RoboDK station: ROXS_2Robots.rdk

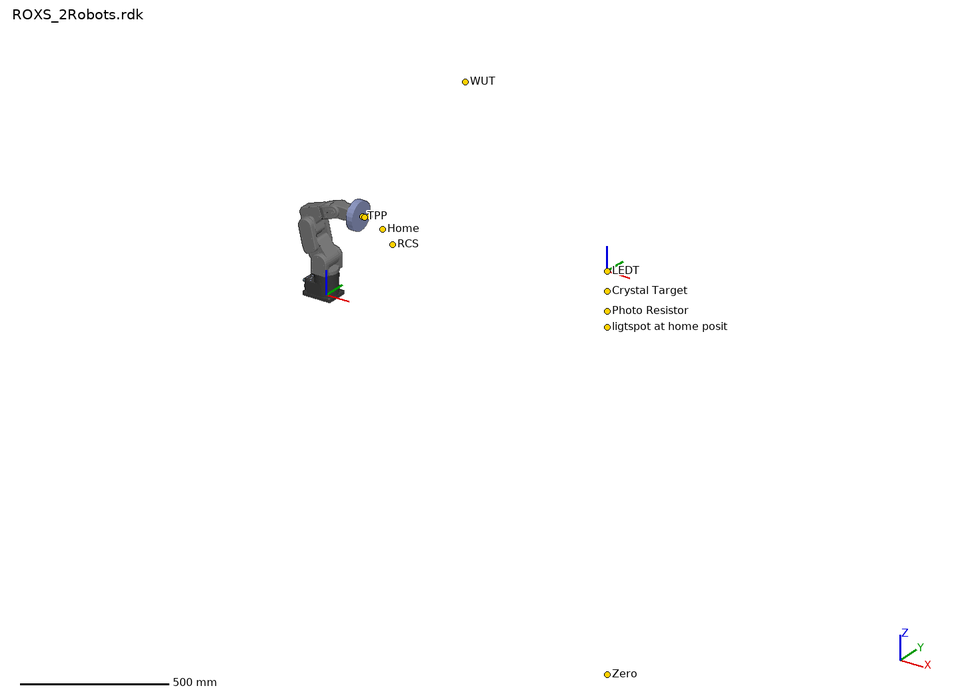
[picture v0: the station drawn from its stored meshes, robots at their saved joint values, targets as dots, program paths as lines]
Station ROXS_2Robots (saved by RoboDK 5.5.2). Poses are relative to the parent item; angles as X-Y-Z fixed-axis rotations.
  - frame LED at (0, 0, 0) mm
    - target Crystal Target (Cartesian target) at (0, 0, -75) mm; joints [-23.128, -26.053, 31.636, -77.168, -23.756, 166.237]
    - target ligtspot at home position (Cartesian target) at (0, 0, -209.55) mm; joints [0, 4.3, -4.481, 0, 0.181, 0]
    - target Zero (Cartesian target) at (0, 0, -1504.55) mm; joints [0, 0, 0, 0, 0, 0] of Mecademic Meca500 R3
    - target WUT (joint target) at (-822.96, 346.08, 338.94) mm, rotated rx -90 ry -86.86 rz -90 deg; joints [0, -22.866, 35.785, 0, -12.919, 0]
    - target Home (Cartesian target) at (-919.2, 0, -101.6) mm, rotated rx 0 ry 90 rz 0 deg; joints [0, 0, 0, 0, 0, 0] of Mecademic Meca500 R3
    - target Zoo wee mama (Cartesian target) at (-982, 12.9, -76.36) mm, rotated rx 0 ry 90 rz 0 deg; joints [12.714, -19.59, 2.794, -37.982, 20.954, -323.903] of Mecademic Meca500 R3
    - target RCS (Cartesian target) at (-950.17, 103.77, -207.82) mm, rotated rx 0 ry 90 rz -5.83 deg; joints [-142.099, -36.249, -124.258, 0, 70.507, -225.257] of Mecademic Meca500 R3
    - target LEDT (Cartesian target) at (0, 0, 0) mm, rotated rx 0 ry 90 rz -5.83 deg; joints [0, -33.951, 22.527, 0, 11.424, 0]
    - target Photo Resistor (Cartesian target) at (0, 0, -150) mm; joints [0, 0, 0, 0, 0, 0]
    - target TPP (Cartesian target) at (-1000, 0, -75) mm, rotated rx 0 ry 90 rz 0 deg; joints [71.078, 20.108, -37.888, -86.424, 78.994, -288.125] of Mecademic Meca500 R3
      - target Bing (Cartesian target) at (75, 0, 1000) mm; joints [0, -10.782, 3.761, 0, 7.021, -360] of Mecademic Meca500 R3
      - target APP (Cartesian target) at (1.62, 1.68, 7.33) mm; joints [0, -22.914, 36.46, 0, -13.546, 0] of Mecademic Meca500 R3
  - Python program Linear Move (listed below)
  - Python program Smart Spiral SSAP (listed below)
  - Python program Set Target Pos (listed below)
  - Python program R Scan (listed below)
  - frame Mecademic Meca500 R3 Base at (-1150, 1.09, -409.6) mm, rotated rx 0 ry 0 rz 0.06 deg
    - robot Mecademic Meca500 R3: 6 axes
        modified DH rows (alpha deg, a mm, theta deg, d mm): 0, 0, 0, 135; -90, 0, -90, 0; 0, 135, 0, 0; -90, 38, 0, 120; 90, 0, 0, 0; -90, 0, 180, 70
        joint limits [-175, -70, -135, -170, -115, -720] to [175, 90, 70, 170, 115, 720]; home [0, 0, 0, 0, 0, 0]; saved at [0.669, -23.965, 5.181, -2.263, 18.798, -357.858]
      - tool CrystalToolSample, TCP at (0, 0, 40.8) mm, size 107.9 x 25.4 x 107.9 mm, geometry from CrystalToolSample.STEP
  - Python program Prog15 (listed below)
  - Python program Prog16 (listed below)
  - Python program SetTarget2 (listed below)
  - Python program R Scan2 (listed below)

--- Python program Linear Move ---
from robodk.robolink import *       # import the robolink library (bridge with RoboDK)
from robodk.robomath import *       # import the robotics toolbox
RDK = Robolink()                    # establish a link with the simulator
robot = RDK.Item('Mecademic Meca500 R3')     # retrieve the robot by name




tool=RDK.Item('CrystalToolSample')
robot.setPoseTool(tool) # Update the TCP

robot.setSpeed(100)  # Set linear speed in mm/s
robot.setJoints([0,0,0,0,0,0])      # set all robot axes to zero



target = RDK.Item('TPP')         # retrieve the Target item
robot.MoveJ(target)                 # move the robot to the target


Final = target.Pose()*transl(0,20,0)
print(target.Pose())

rj=robot.Joints()

print(robot.MoveL_Test(rj,Final))

if robot.MoveL_Test(rj,Final) == 0:         # linear move to the approach position
    robot.MoveL(Final)


print('approach reached')
print('Attempting pose', Final)
#robot.MoveL(pose)

--- Python program Smart Spiral SSAP ---
"""
Created on Thu Jan 19 18:43:18 2023

@author: westj
"""
from robodk.robolink import *       # import the robolink library (bridge with RoboDK)
RDK = Robolink()
from robodk.robomath import *
import math
import numpy as np
import matplotlib.pyplot as plt
import array
import pandas as pd
import requests
import re
from scipy.signal import find_peaks, peak_prominences, savgol_filter
from scipy.stats import linregress
import json
import time
#******CLASSES AND CLASS FUNCTIONS****************************************************************************
class Spiral:
    def __init__(self,x0:float,y0:float,points:float) -> None:
        self.x0=x0 #x offset
        self.y0=y0 #y offset
        self.points=points

    def build(self, radius:float, spacing:float):
        revs=radius/spacing            #calc number of revolutions
        k=spacing/(2*np.pi)
        theta=np.array(np.linspace(0,revs*2*np.pi,self.points)) #how many points and angle coord
        r=k * theta                       #radius coord
        x=(r*np.cos(theta)+self.x0)       #convert to x cartesian
        y=(r*np.sin(theta)+self.y0)       #convert to y cartesian
        return x, y

class Linear:
    def __init__(self,data,points):
        self.data=data #data
        self.points=points #number of points to fit

    def get(self,x):
        peaks= find_peaks(self.data['Intensity'], prominence=[prominence],width=width,height=height)
        IPeaks=peaks[0]
        H=peaks[1]['peak_heights']
        A=[]
        for i in range(len(IPeaks)):
            corr=[IPeaks[i],H[i]]
            A.append(corr)
        SA=sorted(A, key=lambda x: x[1], reverse=True) #sort by peak height largest to smallest
        if len(SA) <= 1:

            E=np.sqrt((Ix-xl)**2+(Iy-yl)**2)
            print('***Linear Translation********************************************************')
            print(Ldata)
            print('_________SSAP Report:_________')
            print('Calculated peak is at',xl,yl)
            print('True peak is at',Ix,Iy)
            print('Error is:',E)
            print('Linear step size is:',step)
            raise Exception("Spiral did not find enough peaks")
        XPP=[]
        YPP=[]
        for i in range(self.points):
            #ICP.append(SA[i][0])
            XPP.append(self.data['X'][SA[i][0]])
            YPP.append(self.data['Y'][SA[i][0]])
        LRR=linregress(XPP,YPP)

        return LRR[0]*x+LRR[1]
    def getC(self,x,xl,yl):
        peaks= find_peaks(self.data['Intensity'], prominence=[prominence],width=width,height=height) #find peaks
        XPP=[xl]  #use origin of previous spiral as a point
        YPP=[yl]
        XPP.append(self.data['X'][peaks[0][0]])
        YPP.append(self.data['Y'][peaks[0][0]])
        LRR=linregress(XPP,YPP) #run regression
        return LRR[0]*x+LRR[1]


    def getSA(self):
        peaks= find_peaks(self.data['Intensity'],prominence=[prominence],width=width,height=height)
        IPeaks=peaks[0]
        H=peaks[1]['peak_heights']
        A=[]
        for i in range(len(IPeaks)):
            corr=[IPeaks[i],H[i]]
            A.append(corr)
        SA=sorted(A, key=lambda g: g[1], reverse=True) #sort by peak height largest to smallest
        return SA,IPeaks

class Webserver:
#webserver returns json string that looks like {"speed":25,"goalpos":140,"zCurrent":140.09935,"PRInt":4,"ledStatus":false,"zero":1}
    def __init__(self,IP,extenstion)->None:
        self.IP=IP #x offset
        self.ex=extenstion #y offset


    def patch(self, obj, value):
        url = "http://" + self.IP + "/" +self.ex #address of server
        obj=str(obj)

        payload = {obj: value} #rewrite the obj to value
        headers = {"Content-Type": "application/json"} #formatting the message as a json string don't change this

        response = requests.patch(url, data=json.dumps(payload), headers=headers) #patch in or change the value

        if response.status_code == 204: #if 204 which is http good patch
            print(obj + "Updated successfully")
        else:
            print(obj + "Error: ", response.status_code)
        return

    def get(self, obj):
        url = "http://" + self.IP + "/" +self.ex #address of server
        obj=str(obj)

        response = requests.get(url)
        if response.status_code == 200:
            value=response.json()[obj]
            print(obj, value)
        else:
           print("Error: ", response.status_code)

        return value


class Intensity: #intensity function is a gaussian curve
    def __init__(self,x0:float,y0:float, mu_x, mu_y, sigma_x, sigma_y):
        self.x0=-x0 #x offset
        self.y0=-y0 #y offset
        self.mu_x=mu_x
        self.mu_y=mu_y
        self.sigma_x=sigma_x #x squish/stretch
        self.sigma_y=sigma_y #y sqush/stretch


    def get(self,x, y): #gaussian curve definition
        I=np.exp(-0.5 * (((x +self.x0- self.mu_x) / self.sigma_x)**2 + ((y+self.y0 - self.mu_y) / self.sigma_y)**2))
        return I

class Photoresistor:
    def __init__(self,url) -> None:
        self.url=url
    def get(self):
        response = requests.get(self.url) #go to webserver under the url of the arduino/photoresistor
        if response.ok: #if we can connect
            value = response.text #screen scrape the web server
            pr=re.findall(r'\d+',value) #take the number off the webserver
            pri=-int(pr[0]) #reverse the sign of the number
            #print('Received value:', value)
            #print('Number', PR)
        else:
            print('Error:', response.status_code)


        return pri

#def Exit_SSAP(Intensity,plateau_size,height):
 #   if len(find_peaks(Intensity,plateau_size=pleatau_size,height=height)[0])>0:
    #    break

#***SPIRAL SCANNING ALIGNMENT PROCEDURE**************************************************************************************************************
#___Initialization______________
xl=0 #starting offset from target for spiral
yl=0
zl=0
Loops=3 #number of loops to run SSAP

robot = RDK.Item('Mecademic Meca500 R3') #define robot
home = RDK.Item('Home') #define robot home
target = RDK.Item('TPP')# retrieve the Target item

tool=RDK.Item('CrystalToolSample')
robot.setPoseTool(tool) # Update the TCP

PR= RDK.Item('Photo Resistor',ITEM_TYPE_TARGET)
X,Y,Z,A,B,C=Pose_2_KUKA(PR.Pose())

IP="192.168.0.99"
ext="values"
ESP=Webserver(IP,ext)

#robot.setSpeed(-1,75)
robot.setSpeed(100)  # Set linear speed in mm/s
robot.MoveJ(home)
print('Robot homed')
robot.MoveJ(target)
print('Robot target approached')

ESP.patch("goalposLED",-Z)
ESP.get("goalposLED")
#ESP.patch("ledStatus",True)
#time.sleep(1)
#ESP.patch("ledStatus",False)
#time.sleep(1)
ESP.patch("ledStatus",True)

for L in range(1,Loops+1):
    if __name__=="__main__":
        print('Starting Spiral '+str(L))

        cur_spiral=Spiral(xl,yl,400) #setting params of the spiral we will be using
        revs=20/L**L
        points=200
        x,y=cur_spiral.build(20/L**2,2/L**2) #build our spiral x y coords
        step=.1/L #linear step size
        zstep=2/L

        Ix=-10
        Iy=10
        TestInt=Intensity(Ix,Iy,0,0,10,10) #set test intensity parameters
        prominence=10
        width=1
        height=50
        plateau_size=2 ############################################
        IAS=10


        #Plot our spiral
        # plt.plot(x, y, color = 'red', marker = "o")
        # plt.axis('equal')
        # plt.show()

    #initialize params
    X=[]
    Y=[]
    Z=[]
    Iv=[]
    Cv=[]

    for i in range(1,len(x)): #loop to get coord and corresponding intensity
        if len(find_peaks(Iv,prominence=[prominence],width=width,height=height)[0])<=0: #check if we found a peak
            if i==len(x):
                print('No peaks found in spiral: Spiral centered')
                coord=(xl,yl,zl)
                robot.MoveJ(target.Pose()*transl(coord))
                raise Exception('Alignment Acheived')
                break
            coord=(x[i],y[i],zl)
            X.append(x[i])
            Y.append(y[i])
            Z.append(0)
            #Ic=PR.get() #get intensity for PR for online run
            Ic=ESP.get("PRInt")
            #Ic=TestInt.get(x[i],y[i]) #test intensity get
            Iv.append(np.array(Ic))

            robot.MoveL(target.Pose()*transl(coord))
            robot.WaitFinished()
        else:
            ps=find_peaks(Iv,prominence=[prominence],width=width,height=height)[0][0]
            fig1 = plt.figure()
            #plt.style.use('seaborn-notebook')
            theta=np.array(np.linspace(0,revs*2*np.pi,points))
            peaks, _ = find_peaks(Iv)

            # height=.1,distance=3,threshold=0.01,
            prominences = peak_prominences(Iv, peaks)[0]
            contour_heights = np.array(Iv)[peaks] - prominences
            plt.plot(Iv)
            plt.plot(peaks, np.array(Iv)[peaks], "x")
            plt.vlines(x=peaks, ymin=contour_heights, ymax=np.array(Iv)[peaks])
            plt.show()

            fig = plt.figure()

            ax = fig.add_subplot(111, projection='3d')
            ax.plot3D(X, Y, Iv)
            ax.plot3D(X[ps], Y[ps], Iv[ps],'x')

            ax.set_xlabel('X axis')
            ax.set_ylabel('Y axis')
            ax.set_zlabel('Z axis')
            plt.show()
            break


    #pandas dictionary
    titled_columns={'X': X,'Y': Y,'Z': Z,
                        'Intensity': Iv}
    data = pd.DataFrame(titled_columns)
    print('Spiral ' +str(L)+ ' Completed')

    if len(find_peaks(data['Intensity'],plateau_size=plateau_size,height=height)[0])>0: #check to see if we are at the peak
        PI=find_peaks(data['Intensity'],plateau_size=plateau_size,height=height)[0]
        xl=data['X'][PI]
        yl=data['Y'][PI]
        coord=(xl,yl,zl)
        print
        robot.MoveL(target.Pose()*transl(coord))
        print('SSAP Complete!')

        break



    CL=Linear(data,2) #current linear line definition


    peaks= find_peaks(data['Intensity'],height=height,prominence=[prominence],width=width)
    IPeaks=peaks[0][0]
    IPeaks=Iv.index(max(Iv))

    xL=data['X'][IPeaks]
    yL=CL.getC(xL,xl,yl) #start y

    Xl=[xL]
    Yl=[yL]

    PRS=data['Intensity'][IPeaks]
    Il=[PRS]

    if  data['X'][IPeaks] > xl:  #find direction to move
        step=step
    else:
        step=-step

    print('Linear move '+str(L)+ ': STARTED')

    #Linear search
    while len(find_peaks(Il,prominence=[prominence],width=width,height=height)[0])<=0: #linear move
        xL=xL+step
        yL=CL.getC(xL,xl,yl)
        PRLT=[]
        for j in range(IAS):
            #PRL=PR.get()
            PRL=ESP.get("PRInt")
            PRLT.append(PRL)

        LI=np.average(PRLT)
        print(PRLT)
        print(LI)
        #PRS=TestInt.get(xL,yL)
        Xl.append(xL)
        Yl.append(yL)
        Il.append(LI)
        print(LI)
        coord=(xL,yL,zl)
        robot.MoveL(target.Pose()*transl(coord))

        if len(find_peaks(-np.array(Il),plateau_size=4,prominence=30)[0])<=0:
            print('Linear moved past alignment')
            break

    print('Linear move '+str(L)+ ': COMPLETED')

    LLdata={'X':Xl,'Y':Yl,'I':Il}
    Ldata=pd.DataFrame(LLdata)

    Lmax_I=Il.index(max(Ldata['I']))
    xl=Xl[Lmax_I]
    yl=Yl[Lmax_I]

    fig = plt.figure()
    #plt.style.use('seaborn-notebook')
    ax = fig.add_subplot(111, projection='3d')
    ax.plot3D(data['X'], data['Y'], data['Intensity'])
    ax.plot3D(data['X'][IPeaks], data['Y'][IPeaks], data['Intensity'][IPeaks],"x")
    ax.plot3D(xl, yl, max(Ldata['I']),"x")
    ax.plot3D(Xl, Yl, Il,'o')

    ax.set_xlabel('X axis')
    ax.set_ylabel('Y axis')
    ax.set_zlabel('Z axis')
    plt.show()

    if len(find_peaks(Ldata['I'],plateau_size=plateau_size,height=height)[0])>0: #check to see if we are at the peak
        PI=find_peaks(Ldata['I'],plateau_size=plateau_size,height=height)[0]
        xl=Ldata['X'][PI]
        yl=Ldata['Y'][PI]
        coord=(xl,yl,zl)
        robot.MoveL(target.Pose()*transl(coord))
        print('SSAP Complete!')
        break


    #Push Pull Search
    IPP=[]
    ZLPP=[]

    for i in range(3):
        coord=(xl,yl,zl)
        ZLPP.append(zl)
        robot.MoveJ(target.Pose()*transl(coord))
        PRPPT=[]
        for j in range(IAS):
            #PRPP=PR.get()
            PRPP=ESP.get("PRInt")
            PRPPT.append(PRPP)
        PPI=np.average(PRPPT)
        IPP.append(PPI)

        zl=zl+(zstep)

    plt.plot(ZLPP,IPP)
    plt.show()

    if IPP.index(max(IPP))>0:
        zstep=zstep
    else:
        zstep=-zstep
    ZLPP=[]
    IPP=[]

    coord=(xl,yl,zl)
    robot.MoveJ(target.Pose()*transl(coord))
    #maybe savitzky golay or moving average filter
    while len(find_peaks(IPP,prominence=5,height=height)[0])<=0: #Push pull
        coord=(xl,yl,zl)
        ZLPP.append(zl)
        robot.MoveL(target.Pose()*transl(coord))
        PRPPT=[]
        for j in range(IAS):
            #PRPP=PR.get()
            PRPP=ESP.get("PRInt")
            PRPPT.append(PRPP)
        PPI=np.average(PRPPT)
        IPP.append(PPI)
        zl=zl+(zstep)


    zl=ZLPP[IPP.index(max(IPP))]


    plt.plot(ZLPP,IPP)
    plt.show()

    #points=100
    #xv,yv=np.meshgrid(np.linspace(-20,20,points),np.linspace(-20,20,points))
    #iv=TestInt.get(xv,yv)
    #ax.plot_surface(xv,yv,iv,alpha=0.5)
    plt.show()
coord=(xl,yl,zl)

ESP.patch("ledStatus",False)
robot.MoveL(target.Pose()*transl(coord))

APP= RDK.Item('APP',ITEM_TYPE_TARGET)
TPP= RDK.Item('TPP',ITEM_TYPE_TARGET)
APP.setParent(TPP)
APP.setPose(Pose(xl,yl,zl,0,0,0))




E=np.sqrt((Ix-xl)**2+(Iy-yl)**2)
print('***Linear Translation********************************************************')
print(Ldata)
print('_________SSAP Report:_________')
print('Calculated peak is at',xl,yl)
print('True peak is at',Ix,Iy)
print('Error is:',E)
print('Linear step size is:',step)

--- Python program Set Target Pos ---
from robolink import *
from robodk import *
import numpy as np
RDK = Robolink()

# Get a reference to the target object
PR = RDK.Item('Photo Resistor',ITEM_TYPE_TARGET)
CT= RDK.Item('Crystal Target',ITEM_TYPE_TARGET)
TPP= RDK.Item('TPP',ITEM_TYPE_TARGET)
RB1 = RDK.Item('Mecademic Meca500 R3 Base',ITEM_TYPE_FRAME)
LED= RDK.Item('LED',ITEM_TYPE_FRAME)


TPP.setParent(LED)
# Define the position of the photoresistor
x=0
y=0
z=-200

#Define offsets of robot 1
x1=-1150
y1=0*25.4
z1=-409.6
a1=0
b1=0
c1=0
tc1=-np.rad2deg(np.arctan(y1/x1))


PR.setPose(Pose(x,y,z,0,0,0))
CT.setPose(Pose(x,y,z/2,0,0,0))
TPP.setPose(Pose(-np.sqrt(1000**2-y1**2),y1,z/2,90,90-tc1,-90))
print(-np.sqrt(1000**2-y1**2))
RB1.setPose(Pose(x1,y1,z1,a1,b1,c1))

reference = TPP.Parent()
print("Target attached to: " + reference.Name())
print("PhotoResistor is at")
print(z)
print("b1 tpp is")
print(tc1)
# You can also move this target to a new reference:
#target.setParent(new_frame)

--- Python program R Scan ---
from robodk.robolink import *       # import the robolink library (bridge with RoboDK)
RDK = Robolink()
from robodk.robomath import *
import math
import numpy as np
import requests
import json

class Webserver:
#webserver returns json string that looks like {"speed":25,"goalpos":140,"zCurrent":140.09935,"PRInt":4,"ledStatus":false,"zero":1}
    def __init__(self,IP,extenstion)->None:
        self.IP=IP #x offset
        self.ex=extenstion #y offset


    def patch(self, obj, value):
        url = "http://" + self.IP + "/" +self.ex #address of server
        obj=str(obj)

        payload = {obj: value} #rewrite the obj to value
        headers = {"Content-Type": "application/json"} #formatting the message as a json string don't change this

        response = requests.patch(url, data=json.dumps(payload), headers=headers) #patch in or change the value

        if response.status_code == 204: #if 204 which is http good patch
            print(obj + "Updated successfully")
        else:
            print(obj + "Error: ", response.status_code)
        return

    def get(self, obj):
        url = "http://" + self.IP + "/" +self.ex #address of server
        obj=str(obj)

        response = requests.get(url)
        if response.status_code == 200:
            value=response.json()[obj]
            print(obj, value)
        else:
           print("Error: ", response.status_code)

        return value



print(0)
# Robot Initialization
robot = RDK.Item('Mecademic Meca500 R3')     # retrieve the robot by name
robot.setSpeed(100)  # Set linear speed in mm/s
tool=RDK.Item('CrystalToolSample')
robot.setPoseTool(tool) # Update the TCP
TPP= RDK.Item('TPP',ITEM_TYPE_TARGET)
LED= RDK.Item('LED',ITEM_TYPE_FRAME)
LEDT= RDK.Item('LEDT',ITEM_TYPE_TARGET)
RCS= RDK.Item('RCS',ITEM_TYPE_TARGET)
PR= RDK.Item('Photo Resistor',ITEM_TYPE_TARGET)
APP= RDK.Item('APP',ITEM_TYPE_TARGET)
#RCS.setParent(LEDT)

#Webserver Initilization
IP="192.168.0.99"
ext="values"
ESP=Webserver(IP,ext)

#Robot Movements
robot.setJoints([0,0,0,0,0,0])      # set all robot axes to zero
print('Homed')

robot.MoveJ(TPP)                 # move the robot to the target
print('Target Approached')


target = RDK.Item('TPP')         # retrieve the Target item
APP.setParent(TPP)
X,Y,Z,A,B,C=Pose_2_KUKA(PR.Pose())
ex,ey,ez,ea,eb,ec=Pose_2_KUKA(APP.Pose())

LEDT.setPose(Pose(0,0,0,0,90,0))


ex=0
ey=0
ez=0
print(ex,ey,ez)
zi=150
zf=200
points=100
PRZ=np.linspace(zi,zf,points)

ESP.patch("ledStatus",True)
for i in range(0,len(PRZ)):
    print(i)
    PR.setParent(LED)
    Z=-1*PRZ[i]
    PR.setPose(Pose(0,0,Z,0,0,0))

    #ESP.patch("speed","100")
    #ESP.patch("goalposLED",abs(Z))

    theta=np.arccos(Z/(2*1000))
    R=Z/2*np.tan(theta)

    #RCS.setPose(Pose(-Z/2+ex,0+ey,-R+ez,0,0,0))

    robot.setPoseTool(tool) # Update the TCP
    coord=(-Z/2+ex,0+ey,-R+ez)





    robot.MoveJ(LEDT.Pose()*transl(coord))
ESP.patch("ledStatus",False)
print('Scan Complete')

--- Python program Prog15 ---
from robodk.robolink import *       # import the robolink library (bridge with RoboDK)
RDK = Robolink()
from robodk.robomath import *
import math
import numpy as np
import requests
import json


print(0)
# Robot Initialization
robot = RDK.Item('Mecademic Meca500 R3')     # retrieve the robot by name
robot.setSpeed(100)  # Set linear speed in mm/s
tool=RDK.Item('CrystalToolSample')
robot.setPoseTool(tool) # Update the TCP


TPP= RDK.Item('TPP',ITEM_TYPE_TARGET)
LED= RDK.Item('LED',ITEM_TYPE_FRAME)
LEDT= RDK.Item('LEDT',ITEM_TYPE_TARGET)
RCS= RDK.Item('Rowland Circle Start',ITEM_TYPE_TARGET)
PR= RDK.Item('Photo Resistor',ITEM_TYPE_TARGET)
APP= RDK.Item('APP',ITEM_TYPE_TARGET)
RCS.setParent(LEDT)
RB1 = RDK.Item('Mecademic Meca500 R3 Base',ITEM_TYPE_FRAME)

TPP.setParent(RB1)

#X,Y,Z,A,B,C=Pose_2_KUKA(PR.Pose())
#ex,ey,ez,ea,eb,ec=Pose_2_KUKA(APP.Pose())
ex=0
ey=0
ez=0

x1=200
y1=0
z1=320
a1=90
b1=90-0
c1=-90

TPP.setPose(Pose(x1,y1,z1,a1,b1,c1))


print(x1,y1,z1)

print(TPP.Pose())

reference = robot.Parent()
print("Target attached to: " + reference.Name())

#for L in range(0,360):
#    TPP.setPose(Pose(x1,y1,z1,a1-L,b1,c1))
robot.MoveJ(TPP.Pose())




print("yay")

--- Python program Prog16 ---
from robodk.robolink import *       # import the robolink library (bridge with RoboDK)

from robodk.robomath import *
RDK = Robolink()
import math
import numpy as np
import requests
import json


print(0)
# Robot Initialization
robot = RDK.Item('Mecademic Meca500 R3')     # retrieve the robot by name
robot.setSpeed(100)  # Set linear speed in mm/s
tool=RDK.Item('CrystalToolSample')
robot.setPoseTool(tool) # Update the TCP


TPP= RDK.Item('TPP',ITEM_TYPE_TARGET)
LED= RDK.Item('LED',ITEM_TYPE_FRAME)
LEDT= RDK.Item('LEDT',ITEM_TYPE_TARGET)
PR= RDK.Item('Photo Resistor',ITEM_TYPE_TARGET)
APP= RDK.Item('APP',ITEM_TYPE_TARGET)
RB1 = RDK.Item('Mecademic Meca500 R3 Base',ITEM_TYPE_FRAME)
BI=RDK.Item('Bing',ITEM_TYPE_TARGET)
TPP.setParent(RB1)
TPP.setParent(LED)
X,Y,Z,A,B,C=Pose_2_KUKA(TPP.Pose())
print(Z)


BI.setParent(TPP)
BI.setPose(Pose(Z,0,1000,0,0,0))



print("yay")

--- Python program SetTarget2 ---
from robolink import *
from robodk import *
import numpy as np
RDK = Robolink()


class Webserver:
#webserver returns json string that looks like {"speed":25,"goalpos":140,"zCurrent":140.09935,"PRInt":4,"ledStatus":false,"zero":1}
    def __init__(self,IP,extenstion)->None:
        self.IP=IP #x offset
        self.ex=extenstion #y offset


    def patch(self, obj, value):
        url = "http://" + self.IP + "/" +self.ex #address of server
        obj=str(obj)

        payload = {obj: value} #rewrite the obj to value
        headers = {"Content-Type": "application/json"} #formatting the message as a json string don't change this

        response = requests.patch(url, data=json.dumps(payload), headers=headers) #patch in or change the value

        if response.status_code == 204: #if 204 which is http good patch
            print(obj + "Updated successfully")
        else:
            print(obj + "Error: ", response.status_code)
        return

    def get(self, obj):
        url = "http://" + self.IP + "/" +self.ex #address of server
        obj=str(obj)

        response = requests.get(url)
        if response.status_code == 200:
            value=response.json()[obj]
            print(obj, value)
        else:
           print("Error: ", response.status_code)

        return value

# Get a reference to the target object
PR = RDK.Item('Photo Resistor',ITEM_TYPE_TARGET)
CT= RDK.Item('Crystal Target',ITEM_TYPE_TARGET)
TPP= RDK.Item('TPP',ITEM_TYPE_TARGET)
RB1 = RDK.Item('Mecademic Meca500 R3 Base',ITEM_TYPE_FRAME)
LED= RDK.Item('LED',ITEM_TYPE_FRAME)
BI=RDK.Item('Bing',ITEM_TYPE_TARGET)

TPP.setParent(LED)
# Define the position of the photoresistor
zPR=-150

#Define offsets of robot 1
x1=-1150
y1=1.09
z1=-409.6
a1=0
b1=0
c1=0.06

tc1=-np.rad2deg(np.arctan(y1/x1))


PR.setPose(Pose(0,0,zPR,0,0,0))
CT.setPose(Pose(0,0,zPR/2,0,0,0))


FD=1000
YLT=0*25.4 #safe distance
bt1=np.rad2deg(np.arcsin(YLT/FD))

XLT=-np.sqrt(FD**2-YLT**2)

TPP.setPose(Pose(XLT,YLT,zPR/2,90,90-bt1,-90))

RB1.setPose(Pose(x1,y1,z1,a1,b1,c1))

BI.setParent(TPP)
BI.setPose(Pose(-zPR/2,0,1000,0,0,0))

--- Python program R Scan2 ---
from robodk.robolink import *       # import the robolink library (bridge with RoboDK)
RDK = Robolink()
from robodk.robomath import *
import math
import numpy as np
import requests
import json

class Webserver:
#webserver returns json string that looks like {"speed":25,"goalpos":140,"zCurrent":140.09935,"PRInt":4,"ledStatus":false,"zero":1}
    def __init__(self,IP,extenstion)->None:
        self.IP=IP #x offset
        self.ex=extenstion #y offset


    def patch(self, obj, value):
        url = "http://" + self.IP + "/" +self.ex #address of server
        obj=str(obj)

        payload = {obj: value} #rewrite the obj to value
        headers = {"Content-Type": "application/json"} #formatting the message as a json string don't change this

        response = requests.patch(url, data=json.dumps(payload), headers=headers) #patch in or change the value

        if response.status_code == 204: #if 204 which is http good patch
            print(obj + "Updated successfully")
        else:
            print(obj + "Error: ", response.status_code)
        return

    def get(self, obj):
        url = "http://" + self.IP + "/" +self.ex #address of server
        obj=str(obj)

        response = requests.get(url)
        if response.status_code == 200:
            value=response.json()[obj]
            print(obj, value)
        else:
           print("Error: ", response.status_code)

        return value



print(0)
# Robot Initialization
robot = RDK.Item('Mecademic Meca500 R3')     # retrieve the robot by name
robot.setSpeed(100)  # Set linear speed in mm/s
tool=RDK.Item('CrystalToolSample')
robot.setPoseTool(tool) # Update the TCP
TPP= RDK.Item('TPP',ITEM_TYPE_TARGET)
LED= RDK.Item('LED',ITEM_TYPE_FRAME)
LEDT= RDK.Item('LEDT',ITEM_TYPE_TARGET)
RCS= RDK.Item('RCS',ITEM_TYPE_TARGET)
PR= RDK.Item('Photo Resistor',ITEM_TYPE_TARGET)
APP= RDK.Item('APP',ITEM_TYPE_TARGET)
#RCS.setParent(LEDT)

#Webserver Initilization
IP="192.168.0.99"
ext="values"
ESP=Webserver(IP,ext)

#Robot Movements
#robot.setJoints([0,0,0,0,0,0])      # set all robot axes to zero
print('Homed')

#robot.MoveJ(TPP)                 # move the robot to the target
print('Target Approached')


target = RDK.Item('TPP')         # retrieve the Target item
APP.setParent(TPP)
LEDT.setPose(Pose(0,0,0,0,90,0))

X,Y,Z,A,B,C=Pose_2_KUKA(PR.Pose())
tx,ty,tz,ta,tb,tc=Pose_2_KUKA(TPP.Pose())
ex,ey,ez,ea,eb,ec=Pose_2_KUKA(APP.Pose())
#tx,ty,tz,ta,tb,tc=Pose_2_KUKA(LEDT.Pose())

LEDT.setPose(LEDT.Pose()*rotx(np.deg2rad(-ta)))
print(ta,tb,tc)
#LEDT.setParent(LED)




print(ex,ey,ez)
zi=150
zf=400
points=300
PRZ=np.linspace(zi,zf,points)

ESP.patch("ledStatus",True)
for i in range(0,len(PRZ)):
    print(i)
    PR.setParent(LED)
    Z=-1*PRZ[i]
    PR.setPose(Pose(0,0,Z,0,0,0))

    ESP.patch("speed","100")
    ESP.patch("goalposLED",abs(Z))
    ESP.get("goalposLED")

    theta=np.arccos(Z/(2*1000))
    R=Z/2*np.tan(theta)

    #RCS.setPose(Pose(-Z/2+ex,0+ey,-R+ez,0,0,0))

    robot.setPoseTool(tool) # Update the TCP
    coord=(-Z/2+ex,0+ey,-R+ez)


    print(coord)

    RCS.setPose(LEDT.Pose()*transl(coord))

    robot.MoveJ(LEDT.Pose()*transl(coord))
    #pause(0.5)
ESP.patch("ledStatus",False)
print('Scan Complete')
